# EPICS autosave request: iocBoot/generic_motors_ioc/dbSave/GS_St_.req
%
% BURT Request File
%
% $(P)GS:St:  GS support
%

file assy.req ASSY=$(P)GS:St
file mtr1.req MTR1=$(P)GS:myw
file mtr1.req MTR1=$(P)GS:mx
file mtr1.req MTR1=$(P)GS:mpt
file drv1.req DRV1=$(P)GS:YW
file drv1.req DRV1=$(P)GS:X
file drv1.req DRV1=$(P)GS:PT
